Staubli VAL3: readStrValue.pgx

public program readStrValue(num x_nCamID (dimensions=1), string x_sCellNumber (dimensions=1), string& x_sValue[] (dimensions=1), bool& x_bError[] (dimensions=1))
  local string l_sCell
  local bool l_bIsOk
begin
  //-----------------------------------------------------------------------
  //Header begin
  //Description of program
  //  Read contents of a cell addressed by col and row from camera' ID.
  //  Returns the contents in value of type string.
  //
  //Input parameters
  //  num x_nCamID :
  //    role : camera's ID
  //  string x_sCellNumber :
  //    role : The column letter and the row number of the cell value to get.
  //    possible values : - column letter : (A to Z)
  //                      - row number : (000 to 399)
  //
  //Output parameters
  //  string x_sValue :
  //    role : contents of cell
  //  bool x_bError :
  //    role : returns true if an error occurred and false otherwise
  //
  //Examples
  //  call readStrValue(nCamID,"D5",l_sValue,x_bError)
  //
  //History
  //  Creation : 19-05-08 - f.Rob
  //Header end
  //-----------------------------------------------------------------------

  nProgram[x_nCamID]=8
  x_bError=true
  // Check format of the cell to read
  call checkCellFormat(x_nCamID,x_sCellNumber,l_bIsOk)
  if l_bIsOk
    call sendCommand(x_nCamID,"GV"+x_sCellNumber,x_bError)
    if !x_bError
      call readSocket(x_nCamID,x_sValue,x_bError)
    else
      x_sValue=""
    endIf
  endIf
end
